PROGRAM TcpServer1Vision
VAR_INPUT
	ServerNetId			: STRING; 	(* Server AmsNetId *)
	ServerAdr 			: STRING;	(* Server IP address *)
	ServerPort 			: UDINT;	(* Server port number *)
END_VAR
VAR_OUTPUT
	busy				: BOOL;
	error				: BOOL;
	errorId				: UDINT;
	bytesReceived		: UDINT;
	
	receiveStruct		: TcpData;	(* Data received *)
	connected 			: BOOL;
END_VAR
VAR
	fbSocketCloseAll 	: FB_SocketCloseAll;
	fbSocketClose 		: FB_SocketClose;
	
	fbSocketListen		: FB_SocketListen;
	fbSocketAccept		: FB_SocketAccept;
	fbSocketReceive		: FB_SocketReceive;
	fbSocketSend 		: FB_SocketSend;
	
	listenerSocket		: T_HSOCKET;
	dataSocket			: T_HSOCKET;
	
	sendQueue 			: TcpDataQueue;
	sendBuffer 			: ARRAY[0..99] OF BYTE;
	
	sendHeartbeats		: BOOL;
	autoDisconnect		: BOOL;
	
	setupStep 			: (CLOSE_CONNECTIONS, CREATE_LISTENER, ACCEPT_CONNECTION, FINISH_SETUP);
	
	setupTimer : TON;
	connectionTimer	: TON;
	heartbeatTimer : TON;
END_VAR
VAR CONSTANT
	connectionTimeout	: TIME := T#30S; //time before connection is closed
	heartbeatInterval	: TIME := T#20S; //heartbeat intervals
	
	incomingHeartbeat	: STRING := 'HEARTBEAT_CLIENT_TO_SERVER';
	outgoingHeartbeat	: STRING := 'HEARTBEAT_SERVER_TO_CLIENT';
END_VAR

blocks();

connected := setup();
IF NOT connected THEN
	RETURN;
END_IF

receive(); //receive in real time

IF autoDisconnect THEN
	autoDisconnectSeq();
ELSE
	connectionTimer.IN := FALSE;
END_IF

IF sendHeartbeats THEN
	sendHeartbeatSeq();
ELSE
	heartbeatTimer.IN := FALSE;
END_IF

send();

METHOD PRIVATE autoDisconnectSeq : BOOL
connectionTimer(IN := , PT := connectionTimeout, Q => , ET => );
connectionTimer.IN := TRUE;

IF connectionTimer.Q THEN
	connectionTimer.IN := FALSE;
	
	closeSocket(dataSocket);
	//closeSocket(listenerSocket);
	
	setupStep := CLOSE_CONNECTIONS;
	RETURN;
END_IF
END_METHOD

METHOD PRIVATE blocks : BOOL
fbSocketClose(
	sSrvNetId:= ServerNetId, 
	hSocket:= dataSocket, 
	bExecute:= , 
	tTimeout:= , 
	bBusy=> busy, 
	bError=> error, 
	nErrId=> errorId);
	
fbSocketCloseAll(
	sSrvNetId:= ServerNetId, 
	bExecute:= , 
	tTimeout:= , 
	bBusy=> , 
	bError=> , 
	nErrId=> );
	
IF fbSocketClose.bExecute OR fbSocketCloseAll.bExecute THEN
	fbSocketClose.bExecute := FALSE;
	fbSocketCloseAll.bExecute := FALSE;
END_IF
	
fbSocketListen(
	sSrvNetId:= ServerNetId, 
	sLocalHost:= ServerAdr, 
	nLocalPort:= ServerPort, 
	bExecute:= , 
	tTimeout:= , 
	bBusy=> busy, 
	bError=> error, 
	nErrId=> errorId, 
	hListener=> listenerSocket);

fbSocketAccept(
	sSrvNetId:= ServerNetId, 
	hListener:= listenerSocket, 
	bExecute:= , 
	tTimeout:= , 
	bAccepted=> , 
	bBusy=> busy, 
	bError=> error, 
	nErrId=> errorId, 
	hSocket=> dataSocket);
	
fbSocketReceive(
	sSrvNetId:= ServerNetId, 
	hSocket:= dataSocket, 
	cbLen:= SIZEOF(receiveStruct), 
	pDest:= ADR(receiveStruct), 
	bExecute:= , 
	tTimeout:= , 
	bBusy=> busy, 
	bError=> error, 
	nErrId=> errorId, 
	nRecBytes=> bytesReceived);
	
fbSocketSend(
	sSrvNetId:= ServerNetId, 
	hSocket:= dataSocket, 
	cbLen:= SIZEOF(sendBuffer), 
	pSrc:= ADR(sendBuffer), 
	bExecute:= , 
	tTimeout:= ,
	bBusy=> busy, 
	bError=> error, 
	nErrId=> errorId);
END_METHOD

METHOD PRIVATE clearBuffer : BOOL
MEMSET(ADR(receiveStruct), 0, SIZEOF(receiveStruct));
END_METHOD

METHOD PRIVATE closeSocket : BOOL
VAR_INPUT
	socket : REFERENCE TO T_HSOCKET;
END_VAR
fbSocketClose.bExecute := TRUE;
fbSocketClose.hSocket := socket;
END_METHOD

METHOD fetch : BOOL
VAR_IN_OUT
	receiverStruct : TcpData;
END_VAR
VAR
	emptyData : TcpData;
END_VAR
fetch := MEMCMP(ADR(receiveStruct), ADR(emptyData), SIZEOF(TcpData)) <> 0; //returns false if no data

receiverStruct := receiveStruct;
receiveStruct := emptyData;
END_METHOD

METHOD queue : BOOL
VAR_INPUT
	data : REFERENCE TO TcpData;
END_VAR
sendQueue.push(data);
END_METHOD

METHOD PRIVATE receive : BOOL
VAR
	heartbeatCheck : STRING;
END_VAR
fbSocketReceive.bExecute := NOT fbSocketReceive.bExecute;
	
MEMCPY(ADR(heartbeatCheck), ADR(receiveStruct), SIZEOF(heartbeatCheck));
IF heartbeatCheck = incomingHeartbeat THEN
	connectionTimer.IN := FALSE;
END_IF
END_METHOD

METHOD PRIVATE send : BOOL
VAR
	polledData : TcpData;
END_VAR
IF NOT fbSocketSend.bBusy THEN
	polledData := sendQueue.poll();
	MEMCPY(ADR(sendBuffer), ADR(polledData), MIN(SIZEOF(polledData), SIZEOF(sendBuffer)));
END_IF

IF NOT BufferIsEmpty(sendBuffer) THEN
	fbSocketSend.bExecute := NOT fbSocketSend.bExecute;
	
ELSE
	fbSocketSend.bExecute := FALSE;
	
END_IF
END_METHOD

METHOD PRIVATE sendHeartbeatSeq : BOOL
VAR
	temp : TcpData;
END_VAR
heartbeatTimer(IN := , PT := heartbeatInterval, Q =>, ET =>);
heartbeatTimer.IN := TRUE;

IF heartbeatTimer.Q THEN
	MEMCPY(ADR(temp), ADR(outgoingHeartbeat), SIZEOF(outgoingHeartbeat));
	queue(temp);
	
	heartbeatTimer.IN := FALSE;
END_IF
END_METHOD

METHOD PRIVATE setup : BOOL
CASE setupStep OF
	CLOSE_CONNECTIONS:
		fbSocketCloseAll( bExecute:= TRUE );
		fbSocketCloseAll( bExecute:= FALSE );
		setupStep := CREATE_LISTENER;
		
	CREATE_LISTENER:
		fbSocketListen.bExecute := TRUE;
		setupStep := ACCEPT_CONNECTION;
		
	ACCEPT_CONNECTION:
		fbSocketListen.bExecute := FALSE;
		IF fbSocketListen.bError THEN
			setupStep := CLOSE_CONNECTIONS;
			RETURN;
			
		ELSIF NOT fbSocketListen.bBusy AND NOT fbSocketListen.bError THEN
			fbSocketAccept.bExecute := FALSE;
			setupTimer(IN:= , PT:= T#500MS, Q=> , ET=> );
			setupTimer.IN := TRUE;
			IF setupTimer.Q THEN
				fbSocketAccept.bExecute := TRUE;
				setupTimer.IN := FALSE;
			END_IF
		
			IF fbSocketAccept.bAccepted THEN
				setupTimer.IN := FALSE;
				setupStep := FINISH_SETUP;
			END_IF
		END_IF
		
		
	FINISH_SETUP:
		setup := TRUE;
		//fbSocketClose(bExecute := TRUE);
END_CASE
END_METHOD

END_PROGRAM

(* stored: Version 1.1.0.1, ProductVersion 3.1.4024.11
   POU TcpServer1Vision: Id {31186d3a-eba3-4199-837d-a55fc3bf8971}, SpecialFunc None
   Folder Monitoring: Id {e6c043a5-b2e8-4d3d-97b2-e0b6fdac7cf9}
   Method autoDisconnectSeq: Id {fa057c82-a854-4418-9eec-f598e1d70696}
   Method blocks: Id {3b065dd9-c535-4aaf-836b-4a7354222d6b}
   Method clearBuffer: Id {e11626cc-d547-4da5-b914-46db9096f4ad}
   Method closeSocket: Id {8abeeb6a-3def-49db-a601-97d4a951adc2}
   Method fetch: Id {c5194247-71cc-491a-bc48-f7fdefcd5cbc}
   Method queue: Id {1f91282a-2bac-4fdd-b9eb-02e7de0408b2}
   Method receive: Id {91b8ab6c-1d5d-4063-8464-d1d9ec08631e}
   Method send: Id {065ebe5c-f528-47e2-bb55-fb2de8f1332e}
   Method sendHeartbeatSeq: Id {46f27e58-d664-4cd0-ad6e-436e818e6c29}
   Method setup: Id {95af496a-6494-483d-8183-1e3d0946c139} *)
